TYPE E_ClientSteps :
(
	CLIENT_STATE_IDLE,
	CLIENT_STATE_CONNECT_START,
	CLIENT_STATE_CONNECT_WAIT,
	CLIENT_STATE_DATAEXCHA_START,
	CLIENT_STATE_DATAEXCHA_WAIT,
	CLIENT_STATE_CLOSE_START,
	CLIENT_STATE_CLOSE_WAIT,
	CLIENT_STATE_ERROR,
	CLIENT_STATE_DATA_ANALYSE
);
END_TYPE

(* stored: Version 1.1.0.1, ProductVersion 3.1.4024.10
   DUT E_ClientSteps: Id {b15045c8-8d19-4f8a-8b2b-37c55796966b} *)
